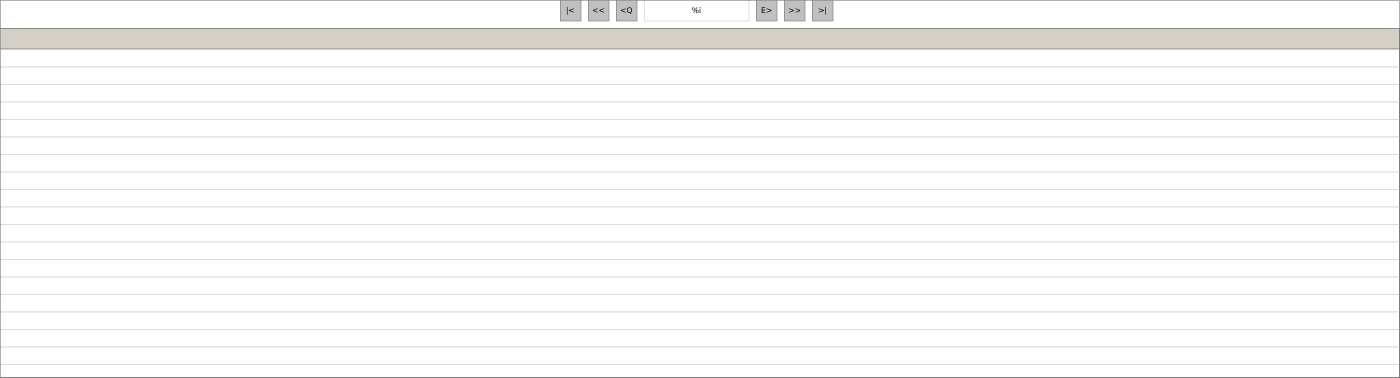
VISUALIZATION LogVisu  // 2000x540
VAR
	selected: INT := 1;
END_VAR
    Table (0,40 2000x500), data array: LogList.list
        p3854506369: LogList.list[INDEX]
        p1137915858: selected
    Textfield (920,0 150x30), "%i", text variable: selected
        OnMouseUp: write the text variable via Default, min 1
    RoundedRectangle (880,0 30x30), "<Q"
        OnMouseUp: execute {
            IF selected > 1 THEN
            	selected := selected - 1;
            END_IF
        }
    RoundedRectangle (1080,0 30x30), "E>"
        OnMouseUp: execute {
            IF selected < 4000 THEN
            	selected := selected + 1;
            END_IF
        }
    RoundedRectangle (840,0 30x30), "<<"
        OnMouseUp: execute {
            IF selected > 25 THEN
            	selected := selected - 24;
            END_IF
        }
    RoundedRectangle (1120,0 30x30), ">>"
        OnMouseUp: execute {
            IF selected < 3975 THEN
            	selected := selected + 24;
            END_IF
        }
    RoundedRectangle (800,0 30x30), "|<"
        OnMouseUp: execute { selected := 1; }
    RoundedRectangle (1160,0 30x30), ">|"
        OnMouseUp: execute { selected := LogList.lastlog; }
    hotkey HotkeyInput Id=481038434304, Key=KeyName=Q, VisuElemId=7
    hotkey HotkeyInput Id=481040531456, Key=KeyName=E, VisuElemId=18
END_VISUALIZATION

(* stored: Version 1.1.0.1, ProductVersion 3.1.4024.12
   Visu LogVisu: Id {c98fb2aa-9752-42c2-b2c3-bf99670ee702} *)
